// TwinCAT 3 PLC project Untitled1
// ProgramVersion: 3.1.4026.14
// libraries:
//   Tc2_Standard, * (Beckhoff Automation GmbH)
//   Tc2_System, * (Beckhoff Automation GmbH)
//   TcUnit, * (www.tcunit.org)
// project tree:
//   / PlcTask.TcTTO
//   POUs/ FC_Add.TcPOU, MAIN.TcPOU
//   TESTs/ FC_Add_Test.TcPOU, PRG_Test.TcPOU
// real-time tasks:
//   TASK PlcTask: cycle T#10ms, priority 20, ADS port 350

CONFIGURATION Untitled1
    RESOURCE PLC ON TwinCAT3
        TASK PlcTask(INTERVAL := T#10ms, PRIORITY := 20);
        PROGRAM MAIN WITH PlcTask : MAIN;
    END_RESOURCE
END_CONFIGURATION

// ---- POUs/MAIN.TcPOU
PROGRAM MAIN
VAR
	a: int ;
END_VAR

Prg_Test();

a:= a+1;

END_PROGRAM

// ---- TESTs/PRG_Test.TcPOU
PROGRAM PRG_Test
VAR
	FC_AddTests : FC_Add_Test;
	
	
END_VAR

TCUnit.RUN();

END_PROGRAM

// ---- TESTs/FC_Add_Test.TcPOU
FUNCTION_BLOCK FC_Add_Test EXTENDS FB_TestSuite
VAR_INPUT
END_VAR
VAR_OUTPUT
END_VAR
VAR
END_VAR

THis^.WhenAAndBArePositveNumbers_ReturnApositivenumber();

METHOD PRIVATE WhenAAndBArePositveNumbers_ReturnApositivenumber
VAR
	a : WORD := 2;
	b : WORD := 3;
	
	actualResult: WORD;
	expectedResult : WORD := 5;
END_VAR
TEST('WhenAAndBArePositveNumbers_ReturnApositivenumber');

//arrange
expectedResult := a+b;

//action
actualResult :=  FC_Add(a,b);

//assert
THIS^.AssertEquals(expectedResult, actualResult,
					Message:= 'The values do not match');

Test_Finished();
END_METHOD

END_FUNCTION_BLOCK

// ---- POUs/FC_Add.TcPOU
FUNCTION FC_Add : WORD
VAR_INPUT
	a :WORD;
	b :WORD;
END_VAR
VAR
END_VAR

FC_Add := a+b;

END_FUNCTION
